// TIA Portal V17 export
// export: Created 2024-06-16T17:47:38.7915191Z, ExportSetting WithDefaults, DisplayName Totally Integrated Automation Portal, DisplayVersion V17, DisplayName TIA Portal Openness, DisplayVersion V17, DisplayName TIA Portal Version Control Interface, DisplayVersion V17, DisplayName STEP 7 Professional, DisplayVersion V17, DisplayName STEP 7 Safety, DisplayVersion V17, DisplayName WinCC Professional, DisplayVersion V17
VAR_GLOBAL   // PLC tag table "St0_In"
   IO_AU_1 AT %I0.0 : Bool;   // Arrêt d'urgence n°1
   IO_AU_2 AT %I0.1 : Bool;   // Arrêt d'urgence n°2
   IO_BP_Rearm AT %I0.2 : Bool;   // Réarmement machine
   IO_Barillet_MP AT %I0.3 : Bool;   // Barillet Métaux Précieux ouvert (MP)
   IO_PorteEntree_Fermee AT %I0.4 : Bool;   // Porte d'entrée : Fermée
   IO_PorteSortie_Fermee AT %I0.5 : Bool;   // Porte de sortie : Fermée
   IO_PorteVision_Fermee AT %I0.6 : Bool;   // Porte maintenance vision façade : Fermée
   IO_PorteArriere_Fermee AT %I0.7 : Bool;   // Portes maitenance arrière machine : Fermée
END_VAR
